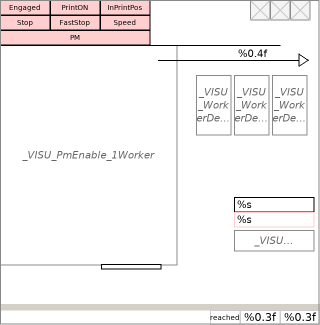
VISUALIZATION _VISU_Pm_WEU_mini_1Worker  // 320x325
VAR_IN_OUT
  mInst : FB_PrintModule_WEU;
END_VAR
    Rectangle (0,40 320x280)
    Frame (234,230 80x21)
        shows _VISU_MarkDetection_Trigger(mInst := mInst.fbMarkDetection)
    Rectangle (234,197 80x15), "%s", tooltip "active camera device", text variable: mInst.fbWorkerCamera._iActiveCam.sName
    Rectangle (234,212 80x15), "%s", tooltip "active camera mode", text variable: mInst.fbWorkerCamera._iActiveCam.eCameraMode, colour toggle: mInst.fbWorkerCamera._bCamValid
    RoundedRectangle (0,304 320x6), colour toggle: mInst.fbView.bMovingInd
    Frame (0,45 177x220)
        shows _VISU_PmEnable_1Worker(mInst := mInst)
        p2738717112: mInst.fbView.zPos_PM
    RoundedRectangle (101,264 60x5), colour toggle: mInst.fbView.bPrintInd[1]
        p2738717112: mInst.fbView.zPos_PM
    Line (0,45) (280,45)
    Rectangle (235,46 80x15), "%0.4f", tooltip "PM position", text variable: mInst._fDistToMasterPm
        OnMouseClick: write the text variable via Default
    Polyline (158,60) (299,60) (299,54) (308,60) (299,66) (299,60)
    RoundedRectangle (280,310 40x15), "%0.3f", tooltip "Target speed", text variable: mInst._pModuleMachineState^.fTargetSpeed
    RoundedRectangle (240,310 40x15), "%0.3f", tooltip "Current Speed", text variable: mInst.fSpeed
    RoundedRectangle (0,30 150x15), "PM", colour toggle: mInst.fbAdsPm.stAds.bI_Enable
    RoundedRectangle (0,0 50x15), "Engaged", colour toggle: mInst._pModuleMachineState^.bEngaged
    RoundedRectangle (50,0 50x15), "PrintON", colour toggle: mInst._pModuleMachineState^.bPrintActivated
    RoundedRectangle (100,0 50x15), "InPrintPos", colour toggle: mInst._pModuleMachineState^.bUnitInPrintPosition
    RoundedRectangle (0,15 50x15), "Stop", colour toggle: NOT mInst._pModuleMachineState^.bStopRequest
    RoundedRectangle (50,15 50x15), "FastStop", colour toggle: NOT mInst._pModuleMachineState^.bFastStopRequest
    RoundedRectangle (100,15 50x15), "Speed", colour toggle: mInst.bSpeedReachedForPrinting
    Image (250,0 20x20), invisible if: NOT mInst._pModuleMachineState^.bSleep, image: sleep_icon
    Image (270,0 20x20), invisible if: NOT mInst._pModuleMachineState^.bShutdown, image: shutdown_icon
    Image (290,0 20x20), invisible if: NOT mInst._pModuleMachineState^.bEStop, image: estop_icon
    RoundedRectangle (210,310 30x15), "reached", tooltip "Target speed reached", colour toggle: mInst._pModuleMachineState^.bTargetSpeedReached
    Frame (234,75 35x60)
        shows _VISU_WorkerDefGrid_small(m_Inst := mInst.fbWorkerDeformation)
    Frame (272,75 35x60)
        shows _VISU_WorkerDefGrid_small(m_Inst := mInst.fbWorkerCamera)
    Frame (196,75 35x60)
        shows _VISU_WorkerDefGrid_small(m_Inst := mInst.fbWorkerPrint[1])
END_VISUALIZATION

(* stored: Version 1.1.0.1, ProductVersion 3.1.4024.11
   Visu _VISU_Pm_WEU_mini_1Worker: Id {344dbd5b-8c55-4692-b99f-6b32f22d15d2} *)
